// SIMATIC S7-200 project (STEP 7-Micro/WIN), CPU 224XP REL 02.01

ORGANIZATION_BLOCK 主程序:OB1
TITLE=程序注释
BEGIN
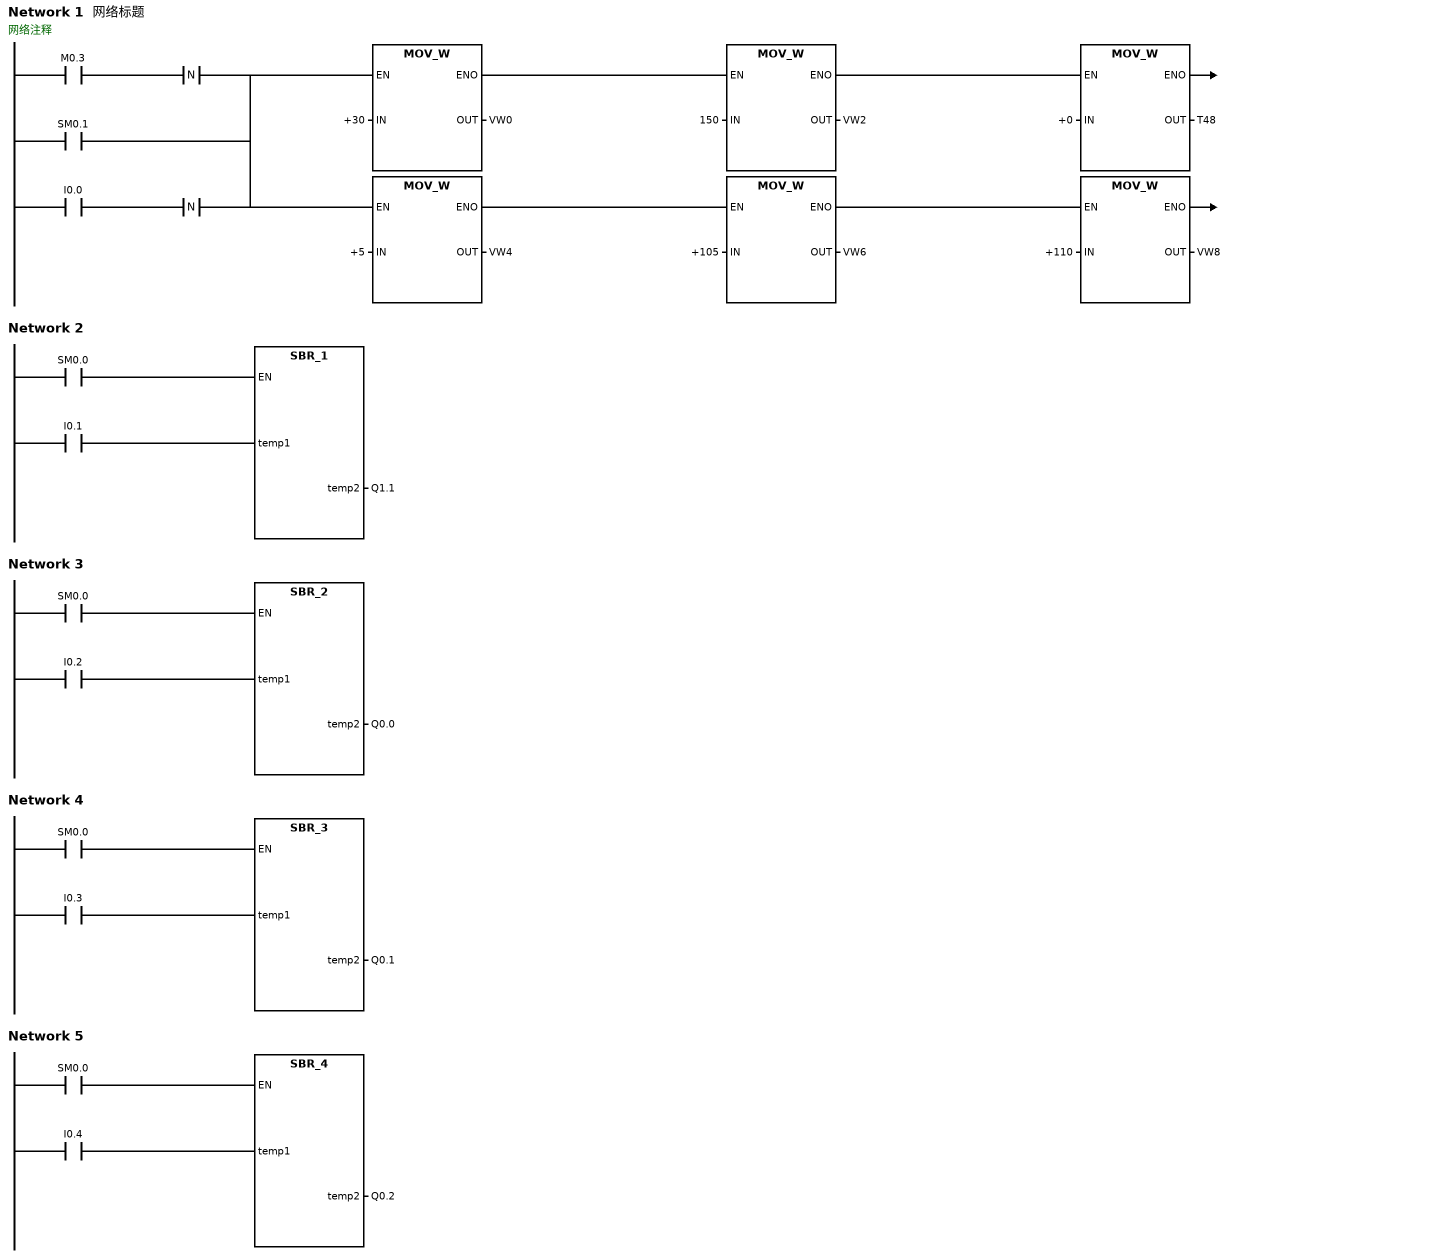
Network 1 // 网络标题
// 网络注释
LD     M0.3
ED
O      SM0.1
LD     I0.0
ED
OLD
LPS
MOVW   +30, VW0
AENO
MOVW   150, VW2
AENO
MOVW   +0, T48
LPP
MOVW   +5, VW4
AENO
MOVW   +105, VW6
AENO
MOVW   +110, VW8
Network 2
LD     SM0.0
=      L60.0
LD     I0.1
=      L63.7
LD     L60.0
CALL   SBR_1:SBR6, L63.7, Q1.1
Network 3
LD     SM0.0
=      L60.0
LD     I0.2
=      L63.7
LD     L60.0
CALL   SBR_2:SBR5, L63.7, Q0.0
Network 4
LD     SM0.0
=      L60.0
LD     I0.3
=      L63.7
LD     L60.0
CALL   SBR_3:SBR4, L63.7, Q0.1
Network 5
LD     SM0.0
=      L60.0
LD     I0.4
=      L63.7
LD     L60.0
CALL   SBR_4:SBR0, L63.7, Q0.2
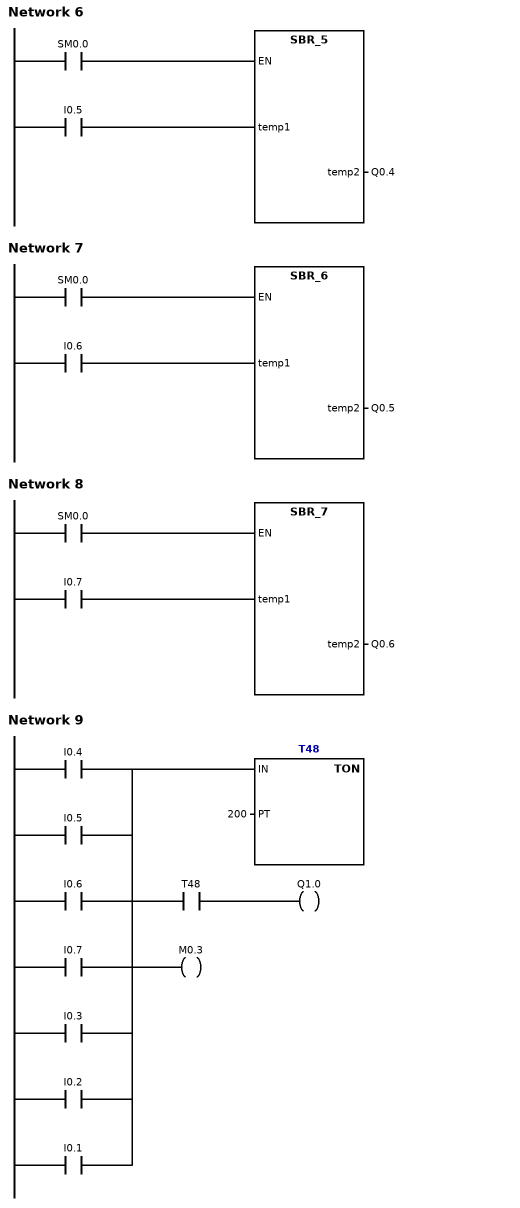
Network 6
LD     SM0.0
=      L60.0
LD     I0.5
=      L63.7
LD     L60.0
CALL   SBR_5:SBR1, L63.7, Q0.4
Network 7
LD     SM0.0
=      L60.0
LD     I0.6
=      L63.7
LD     L60.0
CALL   SBR_6:SBR2, L63.7, Q0.5
Network 8
LD     SM0.0
=      L60.0
LD     I0.7
=      L63.7
LD     L60.0
CALL   SBR_7:SBR3, L63.7, Q0.6
Network 9
LD     I0.4
O      I0.5
O      I0.6
O      I0.7
O      I0.3
O      I0.2
O      I0.1
LPS
TON    T48, 200
A      T48
=      Q1.0
LPP
=      M0.3
END_ORGANIZATION_BLOCK

SUBROUTINE_BLOCK SBR_4:SBR0
TITLE=子程序注释
VAR_INPUT
temp1:BOOL;	// L0.0 
END_VAR
VAR_OUTPUT
temp2:BOOL;	// L0.1 
END_VAR
BEGIN
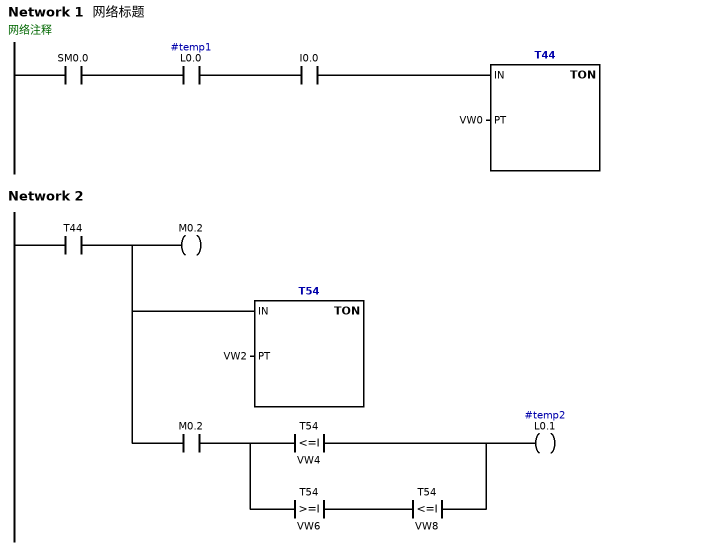
Network 1 // 网络标题
// 网络注释
LD     SM0.0
A      #temp1:L0.0
A      I0.0
TON    T44, VW0
Network 2
LD     T44
=      M0.2
TON    T54, VW2
A      M0.2
LDW<=  T54, VW4
LDW>=  T54, VW6
AW<=   T54, VW8
OLD
ALD
=      #temp2:L0.1
END_SUBROUTINE_BLOCK

SUBROUTINE_BLOCK SBR_5:SBR1
TITLE=
VAR_INPUT
temp1:BOOL;	// L0.0 
END_VAR
VAR_OUTPUT
temp2:BOOL;	// L0.1 
END_VAR
BEGIN
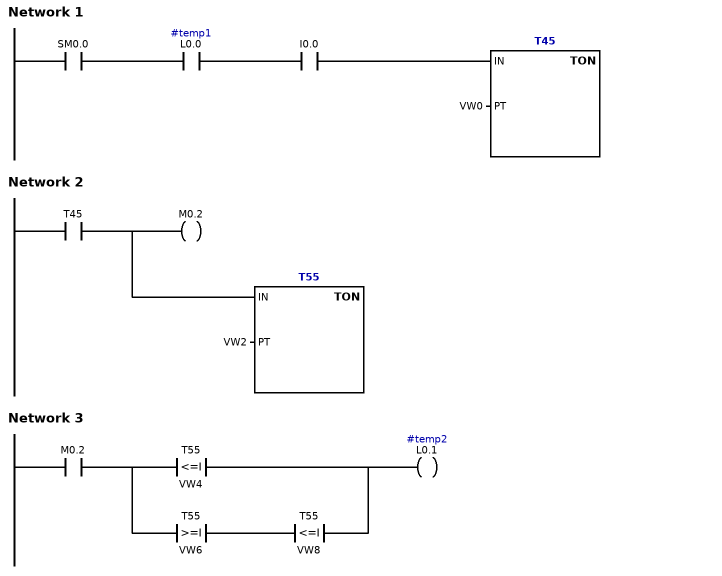
Network 1
LD     SM0.0
A      #temp1:L0.0
A      I0.0
TON    T45, VW0
Network 2
LD     T45
=      M0.2
TON    T55, VW2
Network 3
LD     M0.2
LDW<=  T55, VW4
LDW>=  T55, VW6
AW<=   T55, VW8
OLD
ALD
=      #temp2:L0.1
END_SUBROUTINE_BLOCK

SUBROUTINE_BLOCK SBR_6:SBR2
TITLE=
VAR_INPUT
temp1:BOOL;	// L0.0 
END_VAR
VAR_OUTPUT
temp2:BOOL;	// L0.1 
END_VAR
BEGIN
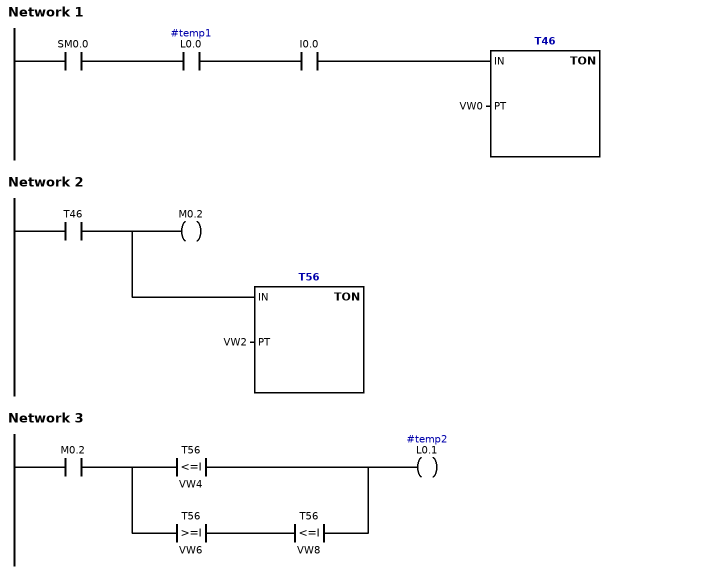
Network 1
LD     SM0.0
A      #temp1:L0.0
A      I0.0
TON    T46, VW0
Network 2
LD     T46
=      M0.2
TON    T56, VW2
Network 3
LD     M0.2
LDW<=  T56, VW4
LDW>=  T56, VW6
AW<=   T56, VW8
OLD
ALD
=      #temp2:L0.1
END_SUBROUTINE_BLOCK

SUBROUTINE_BLOCK SBR_7:SBR3
TITLE=
VAR_INPUT
temp1:BOOL;	// L0.0 
END_VAR
VAR_OUTPUT
temp2:BOOL;	// L0.1 
END_VAR
BEGIN
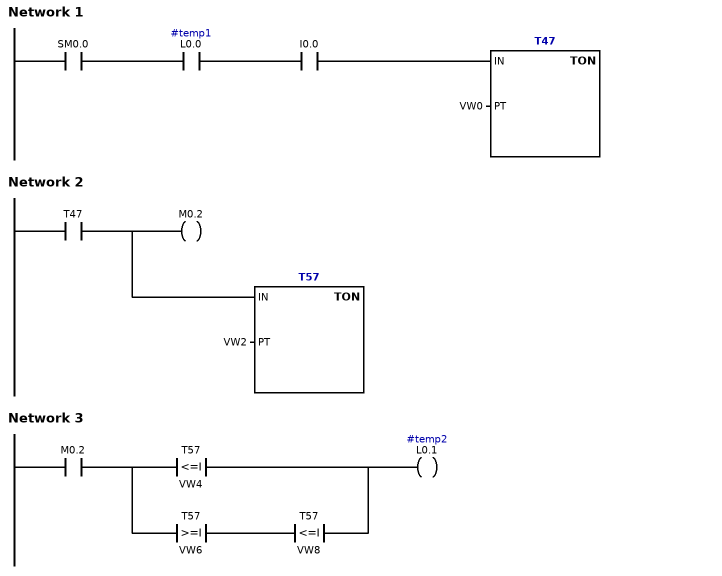
Network 1
LD     SM0.0
A      #temp1:L0.0
A      I0.0
TON    T47, VW0
Network 2
LD     T47
=      M0.2
TON    T57, VW2
Network 3
LD     M0.2
LDW<=  T57, VW4
LDW>=  T57, VW6
AW<=   T57, VW8
OLD
ALD
=      #temp2:L0.1
END_SUBROUTINE_BLOCK

SUBROUTINE_BLOCK SBR_3:SBR4
TITLE=
VAR_INPUT
temp1:BOOL;	// L0.0 
END_VAR
VAR_OUTPUT
temp2:BOOL;	// L0.1 
END_VAR
BEGIN
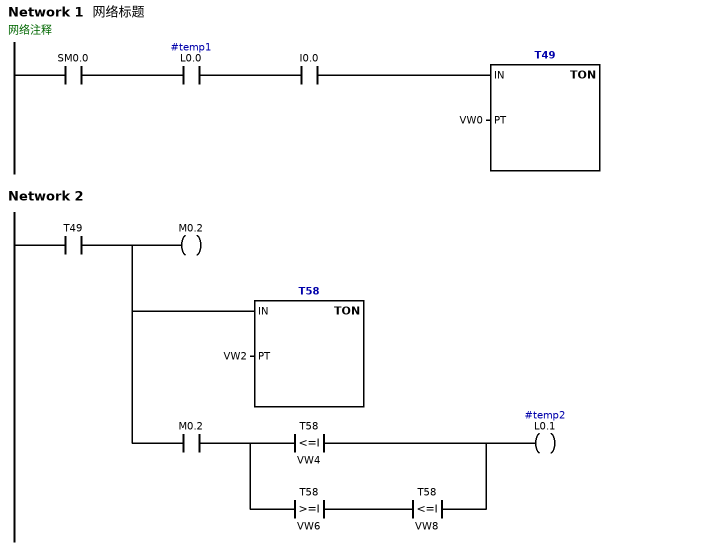
Network 1 // 网络标题
// 网络注释
LD     SM0.0
A      #temp1:L0.0
A      I0.0
TON    T49, VW0
Network 2
LD     T49
=      M0.2
TON    T58, VW2
A      M0.2
LDW<=  T58, VW4
LDW>=  T58, VW6
AW<=   T58, VW8
OLD
ALD
=      #temp2:L0.1
END_SUBROUTINE_BLOCK

SUBROUTINE_BLOCK SBR_2:SBR5
TITLE=
VAR_INPUT
temp1:BOOL;	// L0.0 
END_VAR
VAR_OUTPUT
temp2:BOOL;	// L0.1 
END_VAR
BEGIN
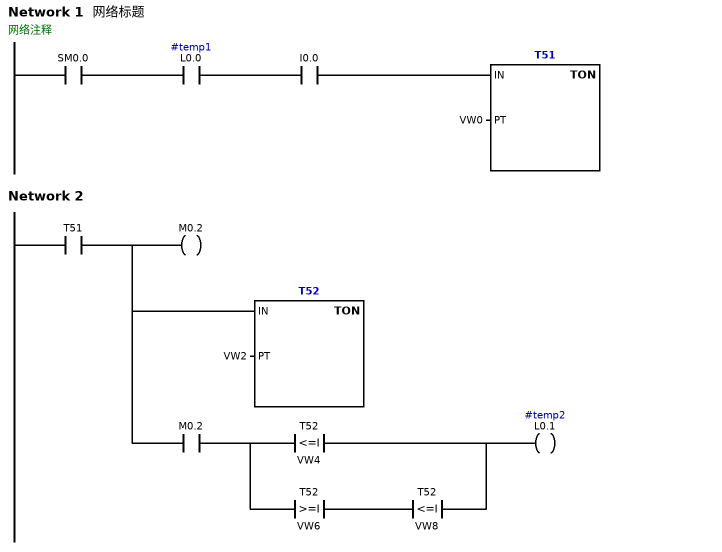
Network 1 // 网络标题
// 网络注释
LD     SM0.0
A      #temp1:L0.0
A      I0.0
TON    T51, VW0
Network 2
LD     T51
=      M0.2
TON    T52, VW2
A      M0.2
LDW<=  T52, VW4
LDW>=  T52, VW6
AW<=   T52, VW8
OLD
ALD
=      #temp2:L0.1
END_SUBROUTINE_BLOCK

SUBROUTINE_BLOCK SBR_1:SBR6
TITLE=
VAR_INPUT
temp1:BOOL;	// L0.0 
END_VAR
VAR_OUTPUT
temp2:BOOL;	// L0.1 
END_VAR
BEGIN
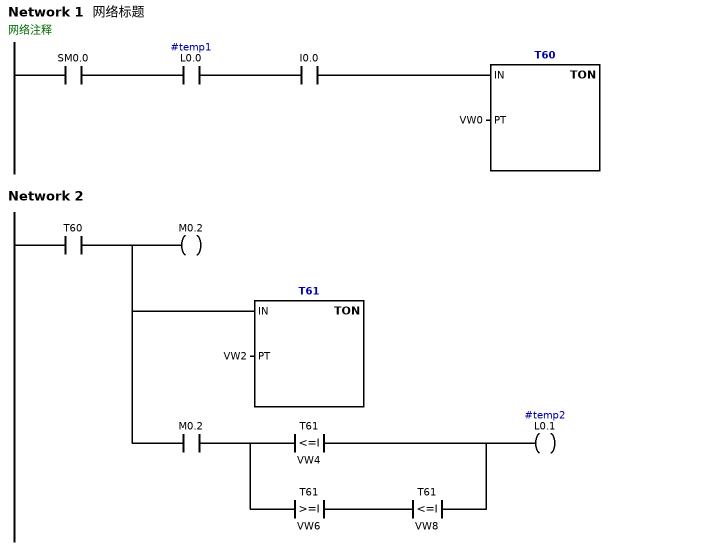
Network 1 // 网络标题
// 网络注释
LD     SM0.0
A      #temp1:L0.0
A      I0.0
TON    T60, VW0
Network 2
LD     T60
=      M0.2
TON    T61, VW2
A      M0.2
LDW<=  T61, VW4
LDW>=  T61, VW6
AW<=   T61, VW8
OLD
ALD
=      #temp2:L0.1
END_SUBROUTINE_BLOCK
